TYPE ST_HMI_USER_MGMT_IN :
STRUCT
	stControlObject					: ST_HMI_GRID_IN;
	sUserManagment_InputString		: STRING;	//Input String Values
	sUserManagment_InputPassword	: STRING;	//Input Password Login
	nUserManagment_InputNumeric		: INT;		//Input Numeric Values
	nUserManagment_InputUserLevel	: INT;		//Input DropDown UserLevel
	stButton_LogOut					: ST_HMI_BUTTON_IN;		//Logout Button
	stButton_LogIn					: ST_HMI_BUTTON_IN;		//Login Button
	stButton_Submit					: ST_HMI_BUTTON_IN;		//Übernehmen Button

	bDeleteUser						: BOOL;
	sCreateDeleteUserName			: STRING;
	sCreateDeleteUserNameConfirm	: STRING;
	sCreateUser_InputPassword		: STRING;	//Input Password Login for create new user
	
	// for Beckhoff HMI UserMgmt:
	iHmiUserLevel					: INT;
END_STRUCT
END_TYPE

(* stored: Version 1.1.0.1
   DUT ST_HMI_USER_MGMT_IN: Id {6e6f38ce-8645-4f10-bb6a-8530f0aa7e73} *)
